# EPICS StreamDevice protocol: proto/mwb_pt100.proto
Terminator = CR;

debug {
	out "%s";
	in "%*#s";
}

getTemperature {
	out "#\$1";
	in ">%f";
}

getModuleName {
	out "$\$1" "M";
	in "!\$1" "%#s";
}

getFirmwareVersion {
	out "$\$1" "F";
	in "!\$1" "%#s";
}
